SUBAPPLICATION AX_OR_3_SPLIT (* 3 unabhaengige AX-Signale je einzeln durchreichen (OUT1/OUT2/OUT3 = IN1/IN2/IN3) UND zusaetzlich gemeinsam ODER-verknuepfen (OUT_OR = IN1 OR IN2 OR IN3) - Sammelstatus 'irgendeiner der 3 ist aktiv', ohne die Einzelsignale zu verlieren. *)
  (* Standard: 61499-2 *)
  (* Version 1.0, 2026-09-17, Franz Höpfinger, Meisterschulen am Ostbahnhof, Ausgelagert aus Baender_Individual_Toggle.SUB (Franz: 'AX_SPLIT_2 AX_SPLIT_3 AX_SPLIT_4 AX_OR_3 in eine SUB auslagern') - dort 3x AX_SPLIT_2 (je 1 Zweig einzeln raus, 1 Zweig in ein gemeinsames AX_OR_3) fuer den Sammelstatus AX_Alle ('ist irgendein Band an'). Wiederverwendbarer, generischer Baustein - nicht baenderspezifisch. *)
  PACKAGE MyLib::sys;
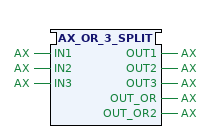
  SOCKETS
    IN1 : adapter::types::unidirectional::AX;
    IN2 : adapter::types::unidirectional::AX;
    IN3 : adapter::types::unidirectional::AX;
  END_SOCKETS
  PLUGS
    OUT1 : adapter::types::unidirectional::AX; (* Durchgereicht von IN1 *)
    OUT2 : adapter::types::unidirectional::AX; (* Durchgereicht von IN2 *)
    OUT3 : adapter::types::unidirectional::AX; (* Durchgereicht von IN3 *)
    OUT_OR : adapter::types::unidirectional::AX; (* IN1 OR IN2 OR IN3 - Sammelstatus *)
    OUT_OR2 : adapter::types::unidirectional::AX;
  END_PLUGS
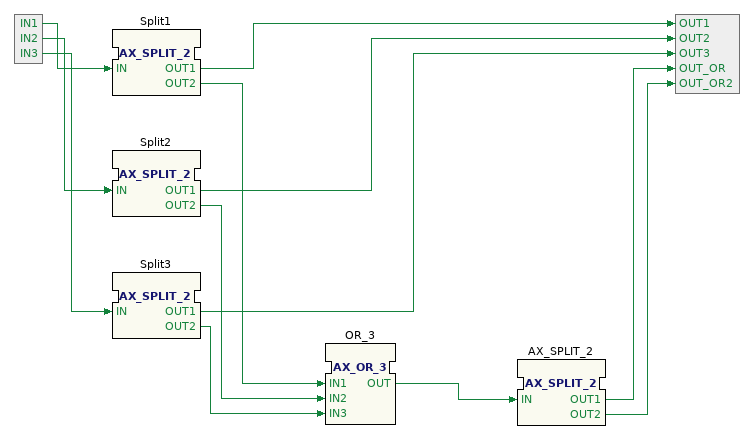
  FBS
    Split1 : adapter::events::unidirectional::AX_SPLIT_2;
    Split2 : adapter::events::unidirectional::AX_SPLIT_2;
    Split3 : adapter::events::unidirectional::AX_SPLIT_2;
    OR_3 : adapter::booleanOperators::AX_OR_3;
    AX_SPLIT_2 : adapter::events::unidirectional::AX_SPLIT_2;
  END_FBS
  ADAPTER_CONNECTIONS
    IN1 TO Split1.IN;
    IN2 TO Split2.IN;
    IN3 TO Split3.IN;
    Split1.OUT1 TO OUT1;
    Split2.OUT1 TO OUT2;
    Split3.OUT1 TO OUT3;
    Split1.OUT2 TO OR_3.IN1;
    Split2.OUT2 TO OR_3.IN2;
    Split3.OUT2 TO OR_3.IN3;
    AX_SPLIT_2.OUT1 TO OUT_OR;
    OR_3.OUT TO AX_SPLIT_2.IN;
    AX_SPLIT_2.OUT2 TO OUT_OR2;
  END_CONNECTIONS
END_SUBAPPLICATION
